FUNCTION_BLOCK PUBLIC EventLogger
VAR
	EventBuffer : ARRAY[1..MAXIMUM_SIZE_OF_EVENT_BUFFER] OF ST_Event; 
	CurrentEventBufferIndex : INT := 0;    
	CurrentEventBufferIndex1 : INT := 1;    
	_PersistentEventStorage : I_PersistentEventStorage; // 声明接口类型的变量
END_VAR
VAR CONSTANT
	MAXIMUM_SIZE_OF_EVENT_BUFFER : INT := 100;
END_VAR

METHOD PUBLIC AddEvent : BOOL
VAR_INPUT
	eEventType : E_EventType;
	eEventSeverity : TcEventSeverity;
	nEventIdentity : UDINT;
	sEventText : STRING(255);
END_VAR
IF NOT IsEventBufferFull() THEN
	CurrentEventBufferIndex := CurrentEventBufferIndex + 1;
	EventBuffer[CurrentEventBufferIndex].eEventType := eEventType;
	EventBuffer[CurrentEventBufferIndex].eEventSeverity := eEventSeverity;
	EventBuffer[CurrentEventBufferIndex].nEventIdentity := nEventIdentity;
	EventBuffer[CurrentEventBufferIndex].sEventText := sEventText;
	UpdateEventTimestampWithSystemTime(stEvent := EventBuffer[CurrentEventBufferIndex]);
	AddEvent := TRUE;
ELSE
	AddEvent := FALSE;
END_IF


//Here we want to store the event persistnetly by a reference
_PersistentEventStorage.StoreEvent(stEvent := EventBuffer[CurrentEventBufferIndex]);
END_METHOD

METHOD FB_init : BOOL
VAR_INPUT
	bInitRetains : BOOL; // if TRUE, the retain variables are initialized (warm start / cold start)
	bInCopyCode : BOOL;  // if TRUE, the instance afterwards gets moved into the copy code (online change)
	iPersistentEventStorage : I_PersistentEventStorage;
END_VAR
_PersistentEventStorage := iPersistentEventStorage; //给EventLogger中的内部变量赋值
END_METHOD

METHOD PRIVATE IsEventBufferFull : BOOL
IF (CurrentEventBufferIndex + 1) > MAXIMUM_SIZE_OF_EVENT_BUFFER THEN
	IsEventBufferFull := TRUE;
ELSE
	ISEventBufferFull := FALSE;
END_IF
END_METHOD

END_FUNCTION_BLOCK

(* stored: Version 1.1.0.1, ProductVersion 3.1.4024.12
   POU EventLogger: Id {3166d354-8b91-4414-9b1a-9d384ad04ae4}, SpecialFunc None
   Method AddEvent: Id {a4ff1506-e495-4043-a98f-591110e3d46d}
   Method FB_init: Id {c023dd39-98cd-4849-be64-ad2548f12aef}
   Method IsEventBufferFull: Id {a4e82661-2f2f-464d-91fb-52707b862608} *)
